{attribute 'linkalways'} 
{attribute 'no_explicit_call' := 'This FB is a CLASS and must be accessed using methods or properties'}
{attribute 'enable_dynamic_creation'}
FUNCTION_BLOCK _ETcVnKnn EXTENDS EnumDatatypeBase
VAR
	localData : ETcVnKnn;
	activeData : REFERENCE TO ETcVnKnn;
	enumBaseDatatype : _UDINT(localData);
END_VAR

METHOD PRIVATE AddLocalEnumeration
VAR_INPUT
	Enumeration : T_MAXSTRING;
	Value : ETcVnKnn;
END_VAR
AddEnumeration(Enumeration, Value);
END_METHOD

PROPERTY PUBLIC Address : PVOID
GET
Address := ADR(activeData);
END_GET
END_PROPERTY

METHOD PUBLIC ClearReference
VAR_INPUT
END_VAR
activeData REF= localData;
SetBaseDatatypeReference();
END_METHOD

METHOD PUBLIC Clone : I_Datatype
VAR
    pClone : POINTER TO _ETcVnKnn;
END_VAR
pClone := __NEW(_ETcVnKnn(InitialValue := Value));
Clone := pClone^;
END_METHOD

METHOD FB_init : BOOL
VAR_INPUT
	bInitRetains : BOOL; // if TRUE, the retain variables are initialized (warm start / cold start)
	bInCopyCode : BOOL;  // if TRUE, the instance afterwards gets moved into the copy code (online change)
	InitialValue : ETcVnKnn;
END_VAR
localData := InitialValue;
AddBaseDatatype(enumBaseDatatype);
ClearReference();

AddLocalEnumeration('TCVN_KNN_CLASSIFIER', ETcVnKnn.TCVN_KNN_CLASSIFIER);
AddLocalEnumeration('TCVN_KNN_NOVELTY_DETECTOR', ETcVnKnn.TCVN_KNN_NOVELTY_DETECTOR);
AddLocalEnumeration('TCVN_KNN_REGRESSOR', ETcVnKnn.TCVN_KNN_REGRESSOR);
END_METHOD

PROPERTY PUBLIC Identifier : T_MAXSTRING
GET
Identifier := 'ETcVnKnn';
END_GET
END_PROPERTY

METHOD IsEnumeratorValueEqual : BOOL
VAR_INPUT
	Enumerator : I_KeyValueForwardEnumerator;
END_VAR
VAR
	storedValue : ETcVnKnn;
END_VAR
IF NOT Enumerator.TryGet(storedValue) THEN
	RETURN;
END_IF

IsEnumeratorValueEqual := storedValue = activeData;
END_METHOD

METHOD PUBLIC MakeReferenceTo
VAR_INPUT
	ReferenceTarget : REFERENCE TO ETcVnKnn;
END_VAR
activeData REF= ReferenceTarget;
SetBaseDatatypeReference();
END_METHOD

METHOD PROTECTED SetBaseDatatypeReference
VAR_INPUT
END_VAR
enumBaseDatatype.MakeReferenceTo(activeData);
END_METHOD

PROPERTY PUBLIC Size : UDINT
GET
Size := SIZEOF(activeData);
END_GET
END_PROPERTY

METHOD TryMakeReferenceTo : BOOL
VAR_INPUT
	Target : I_Datatype;
END_VAR
VAR
	targetAsEnum : I_EnumDatatype;
	pTargetData : POINTER TO ETcVnKnn;
END_VAR
IF NOT Target.TryResolveAsEnumDatatype(targetAsEnum) THEN
	RETURN;
END_IF

IF targetAsEnum.Identifier <> Identifier THEN
	RETURN;
END_IF

pTargetData := Target.Address;
activeData REF= pTargetData^;
SetBaseDatatypeReference();
TryMakeReferenceTo := TRUE;
END_METHOD

PROPERTY PUBLIC Value : ETcVnKnn
GET
Value := activeData;
END_GET
SET
activeData := Value;
END_SET
END_PROPERTY

END_FUNCTION_BLOCK

(* stored: Version 1.1.0.1, ProductVersion 3.1.4024.13
   POU _ETcVnKnn: Id {4eca5e85-c4c5-073d-336f-97bf59fc5749}, SpecialFunc None
   Folder Core: Id {1089ca0c-4069-0e5b-145e-c3afea41f698}
   Folder Protected: Id {89dfd506-5e53-0b76-126d-0c297364f30a}
   Folder Customize: Id {deed7827-8f42-0609-10d3-ae4f0fd481f2}
   Folder Constructor: Id {15cc5049-b073-0130-217a-42a8a634e9da}
   Folder Private: Id {151f09db-cda3-01a7-2728-531598b5199b}
   Folder Protected: Id {0de8942d-64a6-00a1-10e7-dd7168507612}
   Method AddLocalEnumeration: Id {69663167-0bb3-02e4-3ce7-efb5f4e126c8}
   Property Address: Id {88eee2ba-4fff-09b5-19e0-917ffc3643ec}
   Get Get: Id {179dfe30-9d2f-013d-2a17-0ce03505d652}
   Method ClearReference: Id {97d87479-ad0e-02f1-28a7-09aa65faddef}
   Method Clone: Id {f03de18f-4509-074e-2bdc-cd9447398f66}
   Method FB_init: Id {8ce45035-7501-061b-0a21-c3121454515a}
   Property Identifier: Id {bf217c48-ac5c-09dc-25c6-0b696b400371}
   Get Get: Id {0a097cff-1510-0712-1ec7-3849f76d2a45}
   Method IsEnumeratorValueEqual: Id {b87da8dd-1a0f-017f-055e-47f093b69946}
   Method MakeReferenceTo: Id {6bdf91b4-ee30-0453-075d-16dfa507c507}
   Method SetBaseDatatypeReference: Id {d933d899-7537-0159-0ef1-d1b01094a4f4}
   Property Size: Id {dbdd7f6b-eb28-0515-0ca0-4b863bbe6805}
   Get Get: Id {283f3766-9175-07f0-2208-489a02dcd65d}
   Method TryMakeReferenceTo: Id {e1f5ebd3-783a-0e47-1a03-1067a34256c7}
   Property Value: Id {88001680-a8b0-0fa0-37e8-f7c496a06a1f}
   Get Get: Id {b413a931-047d-0485-3e6d-9a3361fc0e9e}
   Set Set: Id {67a90d6f-04be-0226-217e-51959eb6cc95} *)
